FUNCTION_BLOCK timers_ex04
VAR_INPUT
	stand			: Switch_2P;
END_VAR
VAR_OUTPUT
	P1				: DigitalOutput;
	P2				: DigitalOutput;
END_VAR
VAR
	Timer1_ex04		: TON;
	Timer2_ex04		: Tof; 
END_VAR

Timer1_ex04(IN:= stand.position1, PT:= T#10S, Q=> , ET=> );
Timer2_ex04(IN:= P2.On, PT:= T#10S , Q=> , ET=> );
IF stand.position1 THEN
	P1.On();
END_IF
IF Timer1_ex04.Q THEN
	P1.On();
	P2.On();
END_IF
IF Timer2_ex04.Q THEN
	P1.Off();
	P2.Off();
END_IF

END_FUNCTION_BLOCK

(* stored: Version 1.1.0.1
   POU timers_ex04: Id {6e0a85b1-3ae8-40d5-b344-97abe4e87c31}, SpecialFunc None *)
